// Struckig
// Copyright (C) 2022 Stefan Besler

// This program is free software: you can redistribute it and/or modify
// it under the terms of the GNU General Public License as published by
// the Free Software Foundation, either version 3 of the License, or
// (at your option) any later version.

// This program is distributed in the hope that it will be useful,
// but WITHOUT ANY WARRANTY; without even the implied warranty of
// MERCHANTABILITY or FITNESS FOR A PARTICULAR PURPOSE.  See the
// GNU General Public License for more details.
//
// You should have received a copy of the GNU General Public License
// along with THIS PROGRAM.  IF NOT, see <http://www.gnu.org/licenses/>.
{attribute 'qualified_only'}
{attribute 'strict'}
/// Runtime state of the trajectory generator.
TYPE TrajectoryState :
(
  Undefined, //< State has not been initialized yet.
  
  /// The trajectory has reached its final position. For trajectories with a target velocity or/and a target acceleration
  /// there will still be movement.
  Idle,
  
  /// The trajectory is calculated normally
  Busy,
  
  /// An error occured, use [ErrorCode](xref:Struckig.IOtg#ErrorCode) and [ErrorMessage](xref:Struckig.IOtg#ErrorMessage) to get more
  /// information about the error.
  Error
);
END_TYPE

(* stored: Version 1.1.0.1
   DUT TrajectoryState: Id {1b401aa7-ce7a-4de0-8dde-e86175fd1d75} *)
